// TIA Portal V17 export
// export: Created 2025-06-25T13:13:25.6159739Z, ExportSetting WithDefaults, DisplayName Totally Integrated Automation Portal, DisplayVersion V17 Update 8, DisplayName TIA Portal Openness, DisplayVersion V17 Update 8, DisplayName TIA Portal Version Control Interface, DisplayVersion V17, DisplayName STEP 7 Professional, DisplayVersion V17 Update 8, DisplayName STEP 7 Safety, DisplayVersion V17 Update 6, DisplayName WinCC Advanced, DisplayVersion V17 Update 8
DATA_BLOCK "DB_WinCCAlarms"   // DB29
{ S7_Optimized_Access := 'TRUE' }
AUTHOR : Heaten
VERSION : 0.1
// stored: AutoNumber true, DBAccessibleFromOPCUA true, DBAccessibleFromWebserver true, IsOnlyStoredInLoadMemory false, IsRetainMemResEnabled false, IsWriteProtectedInAS false, MemoryReserve 0
   VAR
      "0-System" : Struct
         "0001_WatchdogTimeoutOB1" { S7_SetPoint := 'True'} : "stWinCCAlarm";
         "0003_InitCurrenSettingsFailed" { S7_SetPoint := 'True'} : "stWinCCAlarm";
         "0006_CPUinErrorState" { S7_SetPoint := 'True'} : "stWinCCAlarm";
      END_STRUCT;
      "1-IO" : Struct
         "1001_ConnectionToWinCClost" { S7_SetPoint := 'True'} : "stWinCCAlarm";
         "1002_EmergencyStopActive" { S7_SetPoint := 'True'} : "stWinCCAlarm";
         "1003_SafetyRelayResetFailed" { S7_SetPoint := 'True'} : "stWinCCAlarm";
         "1004_HBL_PS_01_X2" { S7_SetPoint := 'True'} : "stWinCCAlarm";
         "1101_HBL_SC_01_CommError" { S7_SetPoint := 'True'} : "stWinCCAlarm";
         "1102_HBL_SC_02_CommError" { S7_SetPoint := 'True'} : "stWinCCAlarm";
         "1103_HBL_SC_03_CommError" { S7_SetPoint := 'True'} : "stWinCCAlarm";
         "1110_HBL_SC_10_CommError" { S7_SetPoint := 'True'} : "stWinCCAlarm";
         "1121_HBL_SC_01_Tripped" { S7_SetPoint := 'True'} : "stWinCCAlarm";
         "1122_HBL_SC_02_Tripped" { S7_SetPoint := 'True'} : "stWinCCAlarm";
         "1123_HBL_SC_03_Tripped" { S7_SetPoint := 'True'} : "stWinCCAlarm";
         "1130_HBL_SC_10_Tripped" { S7_SetPoint := 'True'} : "stWinCCAlarm";
         "1140_HBL_SC_01_RunFailure" { S7_SetPoint := 'True'} : "stWinCCAlarm";
         "1142_HBL_SC_02_RunFailure" { S7_SetPoint := 'True'} : "stWinCCAlarm";
         "1143_HBL_SC_03_RunFailure" { S7_SetPoint := 'True'} : "stWinCCAlarm";
         "1150_HBL_SC_10_RunFailure" { S7_SetPoint := 'True'} : "stWinCCAlarm";
         "1201_HBL_PT_01_Fault" { S7_SetPoint := 'True'} : "stWinCCAlarm";
         "1202_HBL_PT_02_Fault" { S7_SetPoint := 'True'} : "stWinCCAlarm";
         "1203_HBL_PT_03_Fault" { S7_SetPoint := 'True'} : "stWinCCAlarm";
         "1204_HBL_PT_04_Fault" { S7_SetPoint := 'True'} : "stWinCCAlarm";
         "1205_HBL_TT_05_Fault" { S7_SetPoint := 'True'} : "stWinCCAlarm";
         "1206_HBL_TT_06_Fault" { S7_SetPoint := 'True'} : "stWinCCAlarm";
         "1207_HBL_TT_07_Fault" { S7_SetPoint := 'True'} : "stWinCCAlarm";
         "1208_HBL_TT_08_Fault" { S7_SetPoint := 'True'} : "stWinCCAlarm";
         "1209_HBL_HCV_01_A1_Fault" { S7_SetPoint := 'True'} : "stWinCCAlarm";
         "1210_HBL_TT_10_Fault" { S7_SetPoint := 'True'} : "stWinCCAlarm";
         "1212_HBL_TT_12_Fault" { S7_SetPoint := 'True'} : "stWinCCAlarm";
         "1213_HBL_TT_13_Fault" { S7_SetPoint := 'True'} : "stWinCCAlarm";
         "1214_HBL_TT_14_Fault" { S7_SetPoint := 'True'} : "stWinCCAlarm";
         "1215_HBL_TT_15_Fault" { S7_SetPoint := 'True'} : "stWinCCAlarm";
         "1216_HBL_TT_16_Fault" { S7_SetPoint := 'True'} : "stWinCCAlarm";
         "1217_HBL_TT_17_Fault" { S7_SetPoint := 'True'} : "stWinCCAlarm";
         "1218_HBL_TT_18_Fault" { S7_SetPoint := 'True'} : "stWinCCAlarm";
         "1220_HBL_PT_960_Fault" { S7_SetPoint := 'True'} : "stWinCCAlarm";
         "1221_HBL_PT_05_Fault" { S7_SetPoint := 'True'} : "stWinCCAlarm";
         "1223_HBL_TT_03_Fault" { S7_SetPoint := 'True'} : "stWinCCAlarm";
         "1224_HBL_TT_23_Fault" { S7_SetPoint := 'True'} : "stWinCCAlarm";
         "1225_HBL_TT_24_Fault" { S7_SetPoint := 'True'} : "stWinCCAlarm";
         "1226_HBL_TT_25_Fault" { S7_SetPoint := 'True'} : "stWinCCAlarm";
         "1227_HBL_LT_01_Fault" { S7_SetPoint := 'True'} : "stWinCCAlarm";
         "1228_HBL_TT_21_Fault" { S7_SetPoint := 'True'} : "stWinCCAlarm";
         "1229_HBL_TT_22_Fault" { S7_SetPoint := 'True'} : "stWinCCAlarm";
         "1230_HBL_LT_02_Fault" { S7_SetPoint := 'True'} : "stWinCCAlarm";
         "1231_HBL_HCV_02_A1_Fault" { S7_SetPoint := 'True'} : "stWinCCAlarm";
         "1232_HBL_PT_13_Fault" { S7_SetPoint := 'True'} : "stWinCCAlarm";
         "1233_HBL_TT_20_Fault" { S7_SetPoint := 'True'} : "stWinCCAlarm";
         "1234_HBL_PT_14_Fault" { S7_SetPoint := 'True'} : "stWinCCAlarm";
         "1235_HBL_PT_18_Fault" { S7_SetPoint := 'True'} : "stWinCCAlarm";
         "1236_HBL_PT_19_Fault" { S7_SetPoint := 'True'} : "stWinCCAlarm";
         "1237_HBL_PT_25_Fault" { S7_SetPoint := 'True'} : "stWinCCAlarm";
         "1238_HBL_TT_31_Fault" { S7_SetPoint := 'True'} : "stWinCCAlarm";
         "1239_HBL_TT_33_Fault" { S7_SetPoint := 'True'} : "stWinCCAlarm";
         "1240_HBL_TT_35_Fault" { S7_SetPoint := 'True'} : "stWinCCAlarm";
         "1241_HBL_HCV_01_Fault" { S7_SetPoint := 'True'} : "stWinCCAlarm";
         "1242_HBL_HCV_02_Fault" { S7_SetPoint := 'True'} : "stWinCCAlarm";
         "1243_HBL_PT_07_Fault" { S7_SetPoint := 'True'} : "stWinCCAlarm";
         "1244_HBL_PT_08_Fault" { S7_SetPoint := 'True'} : "stWinCCAlarm";
         "1245_HBL_PT_09_Fault" { S7_SetPoint := 'True'} : "stWinCCAlarm";
         "1246_HBL_PT_10_Fault" { S7_SetPoint := 'True'} : "stWinCCAlarm";
         "1247_HBL_PT_11_Fault" { S7_SetPoint := 'True'} : "stWinCCAlarm";
         "1248_HBL_PT_12_Fault" { S7_SetPoint := 'True'} : "stWinCCAlarm";
         "1249_HBL_PT_15_Fault" { S7_SetPoint := 'True'} : "stWinCCAlarm";
         "1251_HBL_PT_24_Fault" { S7_SetPoint := 'True'} : "stWinCCAlarm";
         "1252_HBL_TT_28_Fault" { S7_SetPoint := 'True'} : "stWinCCAlarm";
         "1253_HBL_TT_29_Fault" { S7_SetPoint := 'True'} : "stWinCCAlarm";
         "1254_HBL_TT_32_Fault" { S7_SetPoint := 'True'} : "stWinCCAlarm";
         "1255_HBL_CT_01_Fault" { S7_SetPoint := 'True'} : "stWinCCAlarm";
         "1256_HBL_CT_02_Fault" { S7_SetPoint := 'True'} : "stWinCCAlarm";
         "1258_HBL_TT_26_Fault" { S7_SetPoint := 'True'} : "stWinCCAlarm";
         "1259_HBL_TT_27_Fault" { S7_SetPoint := 'True'} : "stWinCCAlarm";
         "1260_HBL_FT_01_Fault" { S7_SetPoint := 'True'} : "stWinCCAlarm";
         "1262_HBL_TT_30_Fault" { S7_SetPoint := 'True'} : "stWinCCAlarm";
         "1263_HBL_TT_34_Fault" { S7_SetPoint := 'True'} : "stWinCCAlarm";
         "1264" { S7_SetPoint := 'True'} : "stWinCCAlarm";
         "1265" { S7_SetPoint := 'True'} : "stWinCCAlarm";
         "1266" { S7_SetPoint := 'True'} : "stWinCCAlarm";
         "1267" { S7_SetPoint := 'True'} : "stWinCCAlarm";
         "1268" { S7_SetPoint := 'True'} : "stWinCCAlarm";
         "1269" { S7_SetPoint := 'True'} : "stWinCCAlarm";
         "1270" { S7_SetPoint := 'True'} : "stWinCCAlarm";
         "1271" { S7_SetPoint := 'True'} : "stWinCCAlarm";
         "1272" { S7_SetPoint := 'True'} : "stWinCCAlarm";
         "1273" { S7_SetPoint := 'True'} : "stWinCCAlarm";
         "1274" { S7_SetPoint := 'True'} : "stWinCCAlarm";
         "1275" { S7_SetPoint := 'True'} : "stWinCCAlarm";
         "1276" { S7_SetPoint := 'True'} : "stWinCCAlarm";
         "1277" { S7_SetPoint := 'True'} : "stWinCCAlarm";
         "1278" { S7_SetPoint := 'True'} : "stWinCCAlarm";
         "1279" { S7_SetPoint := 'True'} : "stWinCCAlarm";
         "1280" { S7_SetPoint := 'True'} : "stWinCCAlarm";
         "1281" { S7_SetPoint := 'True'} : "stWinCCAlarm";
         "1282" { S7_SetPoint := 'True'} : "stWinCCAlarm";
         "1283" { S7_SetPoint := 'True'} : "stWinCCAlarm";
         "1284" { S7_SetPoint := 'True'} : "stWinCCAlarm";
         "1285" { S7_SetPoint := 'True'} : "stWinCCAlarm";
         "1286" { S7_SetPoint := 'True'} : "stWinCCAlarm";
         "1287" { S7_SetPoint := 'True'} : "stWinCCAlarm";
         "1288" { S7_SetPoint := 'True'} : "stWinCCAlarm";
         "1289" { S7_SetPoint := 'True'} : "stWinCCAlarm";
         "1290" { S7_SetPoint := 'True'} : "stWinCCAlarm";
         "1291" { S7_SetPoint := 'True'} : "stWinCCAlarm";
         "1292" { S7_SetPoint := 'True'} : "stWinCCAlarm";
         "1293" { S7_SetPoint := 'True'} : "stWinCCAlarm";
         "1294" { S7_SetPoint := 'True'} : "stWinCCAlarm";
         "1295" { S7_SetPoint := 'True'} : "stWinCCAlarm";
      END_STRUCT;
      "2-ProcessValues" : Struct
         "2018" : "stWinCCAlarm";
         "2028" { S7_SetPoint := 'True'} : "stWinCCAlarm";
         "2058" { S7_SetPoint := 'True'} : "stWinCCAlarm";
         "2100" { S7_SetPoint := 'True'} : "stWinCCAlarm";
         "2101" { S7_SetPoint := 'True'} : "stWinCCAlarm";
         "2102" { S7_SetPoint := 'True'} : "stWinCCAlarm";
         "2103" { S7_SetPoint := 'True'} : "stWinCCAlarm";
         "2105" { S7_SetPoint := 'True'} : "stWinCCAlarm";
         "2106" { S7_SetPoint := 'True'} : "stWinCCAlarm";
         "2107" : "stWinCCAlarm";
         "2108" { S7_SetPoint := 'True'} : "stWinCCAlarm";
         "2109" { S7_SetPoint := 'True'} : "stWinCCAlarm";
         "2110" { S7_SetPoint := 'True'} : "stWinCCAlarm";
         "2111" { S7_SetPoint := 'True'} : "stWinCCAlarm";
         "2112" { S7_SetPoint := 'True'} : "stWinCCAlarm";
         "2113" { S7_SetPoint := 'True'} : "stWinCCAlarm";
         "2114" { S7_SetPoint := 'True'} : "stWinCCAlarm";
         "2115" { S7_SetPoint := 'True'} : "stWinCCAlarm";
         "2116" { S7_SetPoint := 'True'} : "stWinCCAlarm";
         "2117" { S7_SetPoint := 'True'} : "stWinCCAlarm";
         "2301_HeatSourceTempDropCritical" { S7_SetPoint := 'True'} : "stWinCCAlarm";
         "2302_HeatSourceTempRiseCritical" { S7_SetPoint := 'True'} : "stWinCCAlarm";
         "2303_SuperheatCompressorHigh" { S7_SetPoint := 'True'} : "stWinCCAlarm";
         "2304_SuperheatCompressorLow" { S7_SetPoint := 'True'} : "stWinCCAlarm";
         "2305_OilFilterDeltaPHigh" { S7_SetPoint := 'True'} : "stWinCCAlarm";
         "2306_OilFilterDeltaPHighHigh" { S7_SetPoint := 'True'} : "stWinCCAlarm";
         "2307_EvaporatorDischargePressureMeanValue" { S7_SetPoint := 'True'} : "stWinCCAlarm";
         "2308_EvaporatorDischargePressureHigh" { S7_SetPoint := 'True'} : "stWinCCAlarm";
         "2309" { S7_SetPoint := 'True'} : "stWinCCAlarm";
      END_STRUCT;
      "3-Control" : Struct
         "3020" : "stWinCCAlarm";
         "3400_HydrolockProtectionActive" : "stWinCCAlarm";
         "3401_DripPanLevelHigh" { S7_SetPoint := 'True'} : "stWinCCAlarm";
      END_STRUCT;
      "4-Communication" : Struct
         dummy : Bool;
      END_STRUCT;
      "5-Auxiliaries" : Struct
         "5000_OilHeatingActivationFailure" : "stWinCCAlarm";
         "5001_OilHeatingDeactivationFailure" { S7_SetPoint := 'True'} : "stWinCCAlarm";
         "5200" : "stWinCCAlarm";
         "5201" { S7_SetPoint := 'True'} : "stWinCCAlarm";
         "5202" { S7_SetPoint := 'True'} : "stWinCCAlarm";
         "5203_CPC_SC_01_CommError" { S7_SetPoint := 'True'} : "stWinCCAlarm";
         "5204_CPC_SC_01_Tripped" { S7_SetPoint := 'True'} : "stWinCCAlarm";
         "5205" { S7_SetPoint := 'True'} : "stWinCCAlarm";
         "5206" { S7_SetPoint := 'True'} : "stWinCCAlarm";
         "5250_SSC_TT_01_Fault" { S7_SetPoint := 'True'} : "stWinCCAlarm";
         "5251_SSC_TT_02_Fault" { S7_SetPoint := 'True'} : "stWinCCAlarm";
         "5252_SSC_TT_03_Fault" { S7_SetPoint := 'True'} : "stWinCCAlarm";
         "5253_SSC_TT_04_Fault" { S7_SetPoint := 'True'} : "stWinCCAlarm";
         "5254_SSC_PIT_01_Fault" { S7_SetPoint := 'True'} : "stWinCCAlarm";
         "5255_SSC_PDT_01_Fault" { S7_SetPoint := 'True'} : "stWinCCAlarm";
         "5256_SSC_LT_01_Fault" { S7_SetPoint := 'True'} : "stWinCCAlarm";
         "5257_SSC_LT_01_Low" { S7_SetPoint := 'True'} : "stWinCCAlarm";
         "5258_SSC_PDT_01_High" { S7_SetPoint := 'True'} : "stWinCCAlarm";
         "5259_SSC_TT_02_High" { S7_SetPoint := 'True'} : "stWinCCAlarm";
         "5260_SSC_TT_03_Low" { S7_SetPoint := 'True'} : "stWinCCAlarm";
         "5261_SSC_PIT_01_Low" { S7_SetPoint := 'True'} : "stWinCCAlarm";
         "5262_DeltaT_ShaftSealHigh" : "stWinCCAlarm";
         "5263_SSC_PIT_01_High" { S7_SetPoint := 'True'} : "stWinCCAlarm";
         "5268_ShaftSealSystemShutdown" { S7_SetPoint := 'True'} : "stWinCCAlarm";
      END_STRUCT;
      "8-Events" : Struct
         "8000_State0_Initialize" : "stWinCCAlarm";
         "8001_State1_Offline" { S7_SetPoint := 'True'} : "stWinCCAlarm";
         "8002_State2_Standby" { S7_SetPoint := 'True'} : "stWinCCAlarm";
         "8003_State3_PrepareStart" { S7_SetPoint := 'True'} : "stWinCCAlarm";
         "8004_State4_Start" { S7_SetPoint := 'True'} : "stWinCCAlarm";
         "8005_State5_Warmup" { S7_SetPoint := 'True'} : "stWinCCAlarm";
         "8006_State6_Running" { S7_SetPoint := 'True'} : "stWinCCAlarm";
         "8007_State7_Stop" { S7_SetPoint := 'True'} : "stWinCCAlarm";
         "8010_Started" : "stWinCCAlarm";
         "8011_Stopped" { S7_SetPoint := 'True'} : "stWinCCAlarm";
         "8014_StartRequestHMI" { S7_SetPoint := 'True'} : "stWinCCAlarm";
         "8015_StartRequestApplication" { S7_SetPoint := 'True'} : "stWinCCAlarm";
         "8018_StopRequestHMI" { S7_SetPoint := 'True'} : "stWinCCAlarm";
         "8019_StopRequestApplication" { S7_SetPoint := 'True'} : "stWinCCAlarm";
         "8020_StopRequestCriticalAlarm" { S7_SetPoint := 'True'} : "stWinCCAlarm";
         "8021_StopRequestControllerFault" { S7_SetPoint := 'True'} : "stWinCCAlarm";
      END_STRUCT;
      "9-Diagnostics" : Struct
         "9021_CondenserBelowSinkTemp" : "stWinCCAlarm";
         "9022_CondensationAboveSinkTemp" { S7_SetPoint := 'True'} : "stWinCCAlarm";
         "9023" { S7_SetPoint := 'True'} : "stWinCCAlarm";
         "9024" { S7_SetPoint := 'True'} : "stWinCCAlarm";
         "9025" { S7_SetPoint := 'True'} : "stWinCCAlarm";
         "9026" { S7_SetPoint := 'True'} : "stWinCCAlarm";
         "9027" { S7_SetPoint := 'True'} : "stWinCCAlarm";
         "9028" { S7_SetPoint := 'True'} : "stWinCCAlarm";
         "9029" { S7_SetPoint := 'True'} : "stWinCCAlarm";
         "9030" { S7_SetPoint := 'True'} : "stWinCCAlarm";
         "9031" { S7_SetPoint := 'True'} : "stWinCCAlarm";
      END_STRUCT;
   END_VAR
BEGIN
END_DATA_BLOCK
